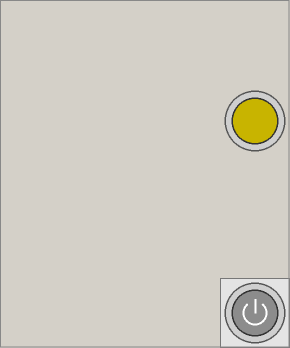
VISUALIZATION HMI  // 290x348
    Lamp1 (220,86 70x70), style: Lamp-Lamp1-Yellow
    PowerSwitch (220,278 70x70), behaviour: TOGGLE, style: Switch-PowerSwitch-Gray
END_VISUALIZATION

(* stored: Version 1.1.0.1, ProductVersion 3.1.4024.12
   Visu HMI: Id {bcde4bf7-5f45-40f0-85f2-1475c27f1c4d} *)
